(* CODESYS project hl3.library
   Title: High level object TwinCAT 3 library
   Version: 0.0.1
   Placeholder: High level object TwinCAT 3 library
   Company: Tomas Rompotl

Project tree, tasks and I/O mapping:
  libraries: Tc2_Standard, * (Beckhoff Automation GmbH); Tc2_System, * (Beckhoff Automation GmbH); Tc3_Module, * (Beckhoff Automation GmbH)
  DataProcessing/
    QuickSort/
      function Partition [ST]
      function QuickSort [ST]
      function Swap [ST]
  DUTs/
  GVLs/
    global variables GVL
  List/
    interface IListItem: data, next
    function block List [ST]: Append
    function block ListOfINT [ST]: Append, FB_init, Get, Insert, IsEmpty, Prepend, Remove, RemoveAll
    function block Node [ST]: data, next
    data type NodeINT
    data type NodeST
  POUs/
    testingUniversalList/
      function block TestFB [ST]
      data type TestStructure
    program ListOfINTTest [ST]
    program ListTest [ST]
    program MAIN [ST]
    program QuickSortTest [ST]: reinit
  Stringify/
    function Stringify [ST]
  VISUs/
*)

// List/NodeINT
{attribute 'enable_dynamic_creation'}
TYPE NodeINT :
STRUCT
	data : INT;
	next : POINTER TO NodeINT;
END_STRUCT
END_TYPE

// List/NodeST
{attribute 'enable_dynamic_creation'}
TYPE NodeST :
STRUCT
	data : ListItem;
	next : POINTER TO Node;
END_STRUCT
END_TYPE

// POUs/testingUniversalList/TestStructure
TYPE TestStructure :
STRUCT
	num : INT;
	str : STRING(80);
	arr : ARRAY[0..3] OF REAL;
END_STRUCT
END_TYPE

// GVLs/GVL
{attribute 'qualified_only'}
VAR_GLOBAL
	vari : int;
END_VAR

// DataProcessing/QuickSort/Partition

// Function used in QuickSort
FUNCTION Partition : INT
VAR_IN_OUT
	ArrayOfREAL			: ARRAY[*] OF REAL; // Partition this array from index nLow to index nHigh
END_VAR
VAR_INPUT
	FirstIndex			: INT; // Starting comparision index
	LastIndex			: INT; // Ending comparision index
END_VAR
VAR
	Pivot				: REAL; // Compared number
	Leftwall			: INT; // New pivot location
	Iterator			: INT; // For iterator variable
END_VAR


Pivot := ArrayOfREAL[LastIndex];
Leftwall := FirstIndex;

FOR Iterator := FirstIndex TO LastIndex - 1 DO
	IF ArrayOfREAL[Iterator] <= Pivot THEN
		Swap(ArrayOfREAL[Iterator], ArrayOfREAL[Leftwall]);
		Leftwall := Leftwall + 1;
	END_IF
END_FOR

Swap(ArrayOfREAL[Leftwall], ArrayOfREAL[LastIndex]);

Partition := Leftwall;

END_FUNCTION

// DataProcessing/QuickSort/Swap

// Swaps values of to variables
FUNCTION Swap
VAR_IN_OUT
	Number1		: REAL;
	Number2		: REAL;
END_VAR
VAR
	Temp		: REAL;
END_VAR


// Just swap pointers
Temp := Number1;
Number1 := Number2;
Number2 := Temp;

END_FUNCTION

// DataProcessing/QuickSort/QuickSort

// Will sort array of REAL using QuickSort algorithm
FUNCTION QuickSort
VAR_IN_OUT
	ArrayOfREALToSort	: ARRAY[*] OF REAL; // Array to sort
END_VAR
VAR_INPUT
	FirstIndex			: INT; // Start index
	LastIndex			: INT; // End index
END_VAR
VAR 
	PivotLocation		: INT; // Partitioning point
END_VAR


IF FirstIndex < LastIndex THEN
	PivotLocation := Partition(ArrayOfREALToSort, FirstIndex, LastIndex);
	QuickSort(ArrayOfREALToSort, FirstIndex, PivotLocation - 1);
	QuickSort(ArrayOfREALToSort, PivotLocation + 1, LastIndex);
END_IF

END_FUNCTION

// List/IListItem
INTERFACE IListItem

PROPERTY data : INT
GET
END_GET
SET
END_SET
END_PROPERTY

PROPERTY next : POINTER TO Node
GET
END_GET
SET
END_SET
END_PROPERTY

END_INTERFACE

// List/Node
{attribute 'enable_dynamic_creation'}
FUNCTION_BLOCK Node IMPLEMENTS IListItem
VAR_IN_OUT
//	data : INT;
//	next : POINTER TO Node;
END_VAR

PROPERTY data : INT
GET
END_GET
SET
END_SET
END_PROPERTY

PROPERTY next : POINTER TO Node
GET
END_GET
SET
END_SET
END_PROPERTY

END_FUNCTION_BLOCK

// List/List
FUNCTION_BLOCK List
VAR_INPUT
END_VAR
VAR_OUTPUT
	count : UINT;
END_VAR
VAR
	head : POINTER TO Node := NULL;
	tail : POINTER TO Node := NULL;
END_VAR


// linked list implementation reference:
// https://www.codesdope.com/blog/article/c-linked-lists-in-c-singly-linked-list/


METHOD Append : REFERENCE TO List
VAR_INPUT
	data : INT;
END_VAR
VAR
	new : POINTER TO Node;
END_VAR

Append REF= THIS^;

new := __NEW(Node);
new^.data := data;
new^.next := NULL;

IF head = NULL THEN
	head := new;
	tail := new;
ELSE
	tail^.next := new;
	tail := tail^.next;
END_IF
count := count + 1;
END_METHOD

END_FUNCTION_BLOCK

// List/ListOfINT

FUNCTION_BLOCK ListOfINT
VAR_INPUT
END_VAR
VAR_OUTPUT
	count : UINT;
END_VAR
VAR
	head : POINTER TO NodeINT := NULL;
	tail : POINTER TO NodeINT := NULL;
END_VAR


// linked list implementation reference:
// https://www.codesdope.com/blog/article/c-linked-lists-in-c-singly-linked-list/


METHOD Append : REFERENCE TO ListOfINT
VAR_INPUT
	data : INT;
END_VAR
VAR
	new : POINTER TO NodeINT;
END_VAR

Append REF= THIS^;

new := __NEW(NodeINT);
new^.data := data;
new^.next := NULL;

IF head = NULL THEN
	head := new;
	tail := new;
ELSE
	tail^.next := new;
	tail := tail^.next;
END_IF
count := count + 1;
END_METHOD


METHOD FB_init : BOOL
VAR_INPUT
	bInitRetains : BOOL; // if TRUE, the retain variables are initialized (warm start / cold start)
	bInCopyCode : BOOL;  // if TRUE, the instance afterwards gets moved into the copy code (online change)
END_VAR
END_METHOD


METHOD Get : INT
VAR_INPUT
	// indexing from end allowed
	// index = 0 returns first element
	// index = 1 returns seconds element
	// index = -1 returns last element
	// index = -2 return before-last element
	index : INT;
END_VAR
VAR
	current : POINTER TO NodeINT := NULL;
	getIndex : INT;
	i : INT;
END_VAR

IF head = NULL THEN
	Get := 0;
	RETURN;
END_IF;

// Calculate actual index in List
getIndex := (count * BOOL_TO_INT(index < 0)) + index;

// Return 0 for invalid indexes
IF 	(getIndex >= count) OR	// Indexing from begin begins with 0
	(getIndex < 0) // Indexing from end begins with -1
THEN
	Get := 0;
	RETURN;
END_IF


current := head;
FOR i := 1 TO getIndex DO // we already got head in previous line, that's why it's from 1
	IF current^.next = NULL THEN
		Get := 0; RETURN;
	END_IF
	current := current^.next;
END_FOR
Get := current^.data;
END_METHOD

// Inserts new element into given index. Negative indexing is supported
METHOD Insert : REFERENCE TO ListOfINT
VAR_INPUT
	(*
		0 = Prepend;
		1 = Insert into second position;
		-2 = Insert into second position from end;
		-1 = Append;
	*)
	index : INT;
	data : INT;
END_VAR
VAR
	new : POINTER TO NodeINT;
	current : POINTER TO NodeINT;
	insertIndex : INT;
	i : INT;
END_VAR

Insert REF= THIS^;

new := __NEW(NodeINT);
new^.data := data;

// Calculate actual index in List
insertIndex := ((count + 1) * BOOL_TO_INT(index < 0)) + index;

IF insertIndex >= count // Index too high -> append to end
THEN
	Append(data);
	RETURN;
ELSIF insertIndex <= 0 // Index too high from the end -> prepend to beginning
THEN
	Prepend(data);
	RETURN;
END_IF

current := head;
FOR i := 1 TO insertIndex - 1 DO
	current := current^.next;
END_FOR
new^.next := current^.next;
current^.next := new;
count := count + 1;
END_METHOD


METHOD IsEmpty : BOOL
VAR_INPUT
END_VAR

IsEmpty := head = NULL;
END_METHOD


// Pushes data to the beginning of the list
METHOD Prepend : REFERENCE TO ListOfINT
VAR_INPUT
	data : INT;
END_VAR
VAR
	new : POINTER TO NodeINT;
END_VAR

Prepend REF= THIS^;

new := __NEW(NodeINT);
new^.data := data;
new^.next := head;

IF head = NULL THEN
	head := new;
	tail := new;
ELSE
	head := new;
END_IF
count := count + 1;
END_METHOD


METHOD Remove : REFERENCE TO ListOfINT;
VAR_INPUT
	index : INT;
END_VAR
VAR
	current : POINTER TO NodeINT := NULL;
	removeIndex : INT;	
	nodeToRemove : POINTER TO NodeINT;
	i : INT;
END_VAR

Remove REF= THIS^;

IF head = NULL THEN
	RETURN;
END_IF;

// Calculate actual index in List
removeIndex := (count * BOOL_TO_INT(index < 0)) + index; 

// Cancel removal for invalid indexes
IF 	(removeIndex >= count) OR // Indexing from begin begins with 0
	(removeIndex < 0) // Indexing from end begins with -1
THEN
	RETURN;
END_IF

IF removeIndex = 0 THEN
	nodeToRemove := head;
	head := head^.next;
ELSE
	current := head;
	FOR i := 1 TO removeIndex - 1 DO
		current := current^.next;
	END_FOR
	nodeToRemove := current^.next;
	current^.next := current^.next^.next;
END_IF
IF nodeToRemove = tail THEN
	tail := current;
END_IF
__DELETE(nodeToRemove);
count := count - 1;
END_METHOD


METHOD RemoveAll : REFERENCE TO ListOfINT
VAR_INPUT
END_VAR

WHILE head <> NULL DO
	Remove(0);
END_WHILE
END_METHOD

END_FUNCTION_BLOCK

// POUs/testingUniversalList/TestFB
FUNCTION_BLOCK TestFB// IMPLEMENTS ITestProps
VAR_INPUT
END_VAR
VAR_OUTPUT
END_VAR
VAR
END_VAR

END_FUNCTION_BLOCK

// POUs/ListOfINTTest
PROGRAM ListOfINTTest
VAR
	listOfINTExample : ListOfINT;
	
	// init
	first : BOOL := TRUE;
	reinit : BOOL;
	
	// insert test
	insertTest : BOOL;
	insertNumber : INT := 42;
	insertIndex : INT := 0;
	
	// remove test
	removeTest : BOOL;
	removeIndex : INT := 0;
	
	// prepend test
	prependTest : BOOL;
	prependData : INT := -10;
	
	// removeAll test
	removeAllTest : BOOL;
	
	// debug
	test : ARRAY[0..30] OF INT;
	
	// hokusy pokusy
	info : __SYSTEM.VAR_INFO;
	
END_VAR

IF first THEN
	first := FALSE;
	listOfINTExample.Append(3);
	listOfINTExample.Append(4);
	listOfINTExample.Append(5).Prepend(2).Prepend(1);
END_IF;
IF reinit THEN
	reinit := FALSE;
	listOfINTExample.FB_init(FALSE, FALSE);
	first := TRUE;
END_IF

IF insertTest THEN
	insertTest := FALSE;
	listOfINTExample.Insert(insertIndex, insertNumber);
END_IF
IF removeTest THEN
	removeTest := FALSE;
	listOfINTExample.Remove(removeIndex);
END_IF
IF removeAllTest THEN
	removeAllTest := FALSE;
	listOfINTExample.RemoveAll();
END_IF


info := __VARINFO(listOfINTExample);
test[0] := listOfINTExample.Get(0);
test[1] := listOfINTExample.Get(1);
test[2] := listOfINTExample.Get(2);
test[3] := listOfINTExample.Get(3);
test[4] := listOfINTExample.Get(4);
test[5] := listOfINTExample.Get(5);
test[6] := listOfINTExample.Get(6);
test[7] := listOfINTExample.Get(7);
test[8] := listOfINTExample.Get(8);
test[9] := listOfINTExample.Get(9);

test[20] := listOfINTExample.Get(-1);
test[21] := listOfINTExample.Get(-2);
test[22] := listOfINTExample.Get(-3);
test[23] := listOfINTExample.Get(-4);
test[24] := listOfINTExample.Get(-5);
test[25] := listOfINTExample.Get(-6);
test[26] := listOfINTExample.Get(-7);
test[27] := listOfINTExample.Get(-8);
test[28] := listOfINTExample.Get(-9);
test[29] := listOfINTExample.Get(-10);

listOfINTExample.count;

END_PROGRAM

// POUs/ListTest
PROGRAM ListTest
VAR
	//testing
	ts : TestStructure;
	tfb : TestFB;
	
	testList : List;
	info : __SYSTEM.VAR_INFO;
END_VAR

info := __VARINFO(tfb);

END_PROGRAM

// POUs/MAIN

PROGRAM MAIN
VAR
	
END_VAR


ListTest();
ListOfINTTest();

QuickSortTest();

END_PROGRAM

// POUs/QuickSortTest

PROGRAM QuickSortTest
VAR
	TestArray0 : ARRAY[0..20] OF REAL := [
		1, 2, 3, 4, 5, 6, 7, 8, 9, 10,
		42, 3.14, 0.618, 1.618, 2.618
	];
	TestArray1 : ARRAY[0..1] OF REAL := [0.1, -0.2];
	
	init : BOOL;
	sort : BOOL;
END_VAR


IF init THEN
	init := FALSE;
	reinit();
END_IF

IF sort THEN
	sort := FALSE;
	QuickSort(TestArray0, 0, 20);
	QuickSort(TestArray1, 0, 1);
END_IF


METHOD reinit : BOOL
VAR_INPUT
END_VAR
VAR CONSTANT
	Array0 : ARRAY[0..20] OF REAL := [
		1, 2, 3, 4, 5, 6, 7, 8, 9, 10,
		42, 3.14, 0.618, 1.618, 2.618
	];
	Array1 : ARRAY[0..1] OF REAL := [0.1, -0.2];
END_VAR

TestArray0 := Array0;
TestArray1 := Array1;
END_METHOD

END_PROGRAM

// Stringify/Stringify
FUNCTION Stringify : STRING
VAR_INPUT
	info : __SYSTEM.VAR_INFO;
//	another : INT;
END_VAR
VAR
//	info : __SYSTEM.VAR_INFO;
END_VAR

//info := __VARINFO(data);
Stringify := info.Symbol;

END_FUNCTION
